(* CoDeSys 2.3 export: SESH_CODESYS.EXP *)
(* Libraries: C:\Program Files (x86)\WAGO Software\CoDeSys V2.3\Targets\WAGO\Libraries\POWER_MEASUREMENT\PowerMeasurement_494_02.lib 7.10.15 13:30:30, Iecsfc.lib 16.5.13 14:00:50, mod_com.lib 16.5.13 14:00:50, Modb_l05.lib 22.4.13 12:50:12, SerComm.lib 16.5.13 14:00:50, Serial_Interface_01.lib 22.4.13 12:50:14, Standard.lib 20.5.14 08:13:26, SYSLIBCALLBACK.LIB 16.5.13 14:00:50, SysLibFile.lib 16.5.13 14:00:50, SysLibSem.lib 16.5.13 14:00:50, SysLibSockets.lib 22.5.14 16:16:32, SysLibTime.lib 16.5.13 14:00:48, Wago_MBCFG_COMMON_01.lib 5.12.13 11:10:18, Wago_MBCFG_SERIAL_01.lib 17.9.14 14:24:36, WagoLibMySQL_03.lib 23.7.14 09:13:36, WagoLibSHA1.lib 19.9.11 08:14:42 *)

(* PLC configuration (modules and I/O channels)
PLC Configuration [Root] node -1, in %IB0 out %QB0
  K-Bus [K_Bus] node 0, in %IB0 out %QB0 {param 201019000 = 1; param 201019001 = 10000; param 201019002 = 0; param 201019003 = 1}
    0750-0652#24 RS-232/RS-485 Interface adjustable (24 Bytes) [Type_30_1_Channels] node 0, in %IB120 out %QB120
      AT %IB0 [BYTEOnB_I] First Byte of 24
      AT %QB0 [BYTEOnB_Q] First Byte of 24
    0750-0652#24 RS-232/RS-485 Interface adjustable (24 Bytes) [Type_30_1_Channels] node 1, in %IB120 out %QB120
      AT %IB24 [BYTEOnB_I] First Byte of 24
      AT %QB24 [BYTEOnB_Q] First Byte of 24
    0750-0652#24 RS-232/RS-485 Interface adjustable (24 Bytes) [Type_30_1_Channels] node 2, in %IB144 out %QB144
      AT %IB48 [BYTEOnB_I] First Byte of 24
      AT %QB48 [BYTEOnB_Q] First Byte of 24
    0750-0494 3-phase PoM480/ 1A [Type_58_1_Channels] node 3, in %IB168 out %QB168
      AT %IW36 [WORDOnW_I] Status Word
      AT %IW37 [WORDOnW_I] Status Word 1
      AT %IW38 [WORDOnW_I] Status Word 2
      AT %IW39 [WORDOnW_I] Status Word 3
      AT %ID20 [DWORDOnD_I] process value 1
      AT %ID21 [DWORDOnD_I] process value 2
      AT %ID22 [DWORDOnD_I] process value 3
      AT %ID23 [DWORDOnD_I] process value 4
      AT %QW36 [WORDOnW_Q] Control Word
      AT %QW37 [WORDOnW_Q] Control Word 1
      AT %QW38 [WORDOnW_Q] Control Word 2
      AT %QW39 [WORDOnW_Q] Control Word 3
    0750-0494 3-phase PoM480/ 1A [Type_58_1_Channels] node 4, in %IB192 out %QB192
      AT %IW48 [WORDOnW_I] Status Word
      AT %IW49 [WORDOnW_I] Status Word 1
      AT %IW50 [WORDOnW_I] Status Word 2
      AT %IW51 [WORDOnW_I] Status Word 3
      AT %ID26 [DWORDOnD_I] process value 1
      AT %ID27 [DWORDOnD_I] process value 2
      AT %ID28 [DWORDOnD_I] process value 3
      AT %ID29 [DWORDOnD_I] process value 4
      AT %QW48 [WORDOnW_Q] Control Word
      AT %QW49 [WORDOnW_Q] Control Word 1
      AT %QW50 [WORDOnW_Q] Control Word 2
      AT %QW51 [WORDOnW_Q] Control Word 3
    0750-0483 2 AI 0-30V DC Differential Measurement Input [Type_8_2_Channels] node 5, in %IB216 out %QB216
      AT %IW60 [WORDOnW_I] Ch_1 Input word
      AT %IW61 [WORDOnW_I] Ch_2 Input word
    0750-0513/0000-0001 2 DO 250V AC 2.0A Rel 2NO (PotFree) [Type_10_2_Channels] node 6, in %IB124 out %QB120
      AT %QX60.0 [BOOLOnX_Q] Ch_1 Digital output
      AT %QX60.1 [BOOLOnX_Q] Ch_2 Digital output
  Modbus variables [PFC200MODBUS] node 1, in %IB0 out %QB0 {param 2010330101 = 1; param 2010330102 = 1; param 2010330201 = 1; param 2010330202 = 502; param 2010330203 = 600; param 2010330301 = 1; param 2010330302 = 502; param 2010330401 = 0; param 2010330402 = 1; param 2010330403 = 5000; param 2010330404 = 0; param 2010330405 = 115200; param 2010330406 = 1; param 2010330407 = 1; param 2010330408 = 0; param 2010330409 = 0}
  Modbus-Master [MB_MASTER] node 2, in %IB0 out %QB0
*)

(* Task configuration *)
TASK MYSQL_Logging (PRIORITY := 29, INTERVAL := T#1s0ms);
Main_logger();
END_TASK
TASK MB_RTU_MASTER_TASK (PRIORITY := 30, INTERVAL := T#5ms);
MBCFG_ModbusSlave();
END_TASK

(* Global variable list: Global_Variables *)
VAR_GLOBAL

	gv_sFilePath: STRING;
	gv_iBuffCounter			:INT := 0; (* counter for  buffer*)
	gv_iBuffPointer			:INT := 0; (* pointer  for  buffer*)
	gv_Buffer					:ARRAY[0..gc_MaxBufferSize] OF DataPoint; (*In memory buffer of failed message attempts*)
	gv_isGenSetON                 :BOOL := FALSE;
	gv_DCGenCycleCount     : INT :=0 ;
	gv_statusRELAY1 AT %QX60.0: BOOL;
	gv_statusRELAY2 AT %QX60.1: BOOL;

END_VAR
VAR_GLOBAL CONSTANT

	(* Site specific variables*)
	gc_iSiteCode: INT := 1000; (*1000 is code for Nyange this needs to be somehow made dynamic and unique for each site*)


	MAX_ROWS : WORD := 30; (* Array size for converted table data *)

	gcMySql_iSqlUpperBound: INT := 29; (* Defines the upper bound of "asSqlStatement",
				used by function blocks "MySql_ExecSql" and "MySql_Query" 
				to provide an SQL statement as "ARRAY [0..UpperBound] OF STRING(Size)".
	*)

	gcMySql_iSqlLength: INT := 370; (* Defines the size in byte of an array element
				of "asSqlStatement", used by function blocks "MySql_ExecSql" and "MySql_Query" 
				to provide an SQL statement as "ARRAY [0..UpperBound] OF STRING(Size)".
	*)
	raw_SQL_STR_LENGTH: INT := 350;

	(* MYSQL configs *)
	gc_sHost : STRING := '### your mysql server address here';  (*'application.dyndns.info';*)
	gc_uiPort : UINT := 3306;
	gc_sUser : STRING := '### your mysql server username ';
	gc_sPwd : STRING := '### your mysql password';
	gc_sDB : STRING := '### your MYSQL database';   	(* Optional - Name of database instance to connect to *)
	gc_sTable:STRING := '### your MYSql table' ;

	(* CSV Writing/Logging parameters*)
	gc_xWriteToSD: BOOL := TRUE;

	iMaxParams			:INT:=5;(* Number of Parameters per File *)
	gc_ParameterCount	:INT:=1;(* Number of Values per Parameter *)
	gc_RawDataSize		:UINT:=500; (* Raw data size for reading in file ASCII *)
	gc_MaxBufferSize 	       :INT := 5000; (*number of items to hold in memory*)
	gc_sFileName		: STRING := 'buffer.csv'; (* Working Filename   Complete path + filename *)

	(* Logging constants*)
	gc_LogInterval             :TIME := T#10s;
	gc_iTotalParams		:INT := 18;

	(* generator constants*)
	gc_DCVoltageGenSetON :REAL := 24; (*make this a bit higher tha load shedding time*)
	gc_DCVoltageGenSetOFF :REAL := 26; (*make this estimate soc %80*)

	(*how many cycles do we wait before we trigger the genset need to calculate based no cycletime *gc_DCGenCycleCount = total_seconds  *)
	gc_DCGenCycleCount       :INT := 40;

END_VAR

(* Data type *)
TYPE DataPoint :
	STRUCT
		(*Common variables*)
		iSiteCode:INT;
		timeStamp: STRING;

		(*AC Variables*)
		rTotalActivePower:REAL;
		rTotalReactivePower:REAL;
		rTotalApparentPower:REAL;
	      rTotalPowerFactorPF:REAL;
		rTotalActiveEnergy:REAL;
		rTotalReactiveEnergy:REAL;
		rTotalApparentEnergy:REAL;
		xRotatingField:BOOL;
		arFrequency_1:REAL;
		arVoltage_L_N_1:REAL;
		arCurrent_1:REAL;
		arFrequency_2:REAL;
		arVoltage_L_N_2:REAL;
		arCurrent_2:REAL;
		arFrequency_3:REAL;
		arVoltage_L_N_3:REAL;
		arCurrent_3:REAL;

		(* DC Variables *)
		DCV1 :REAL;
		DCV2 :REAL;
		DCPower1: REAL;
		DCPower2: REAL;
		DCCurr1 : REAL;
		DCCurr2 : REAL;


		END_STRUCT
END_TYPE

(* Data type *)
TYPE RowData :
  STRUCT
  	dtDt 		: DT; 		(* Table field "timestamp" 	- MySql_Datatype "datetime" 	*)
  	asString 	: ARRAY [0..9] OF STRING(255);	(* Table fields "s0"-"s9" MySql_Datatype "varchar(255)" 	*)
  END_STRUCT
END_TYPE

(* Data type *)
TYPE TableData :
  STRUCT
	xValid : BOOL;
	iRowCount : INT;
	astRow : ARRAY [0..gcMySql_dwMaxRowCount] OF RowData;
  END_STRUCT
END_TYPE

(* Data type *)
TYPE typCSV :
STRUCT
	sDescription	:STRING;
	Parameter		:ARRAY[1..gc_ParameterCount] OF REAL;
END_STRUCT
END_TYPE

(* POU Main_logger, ST *)
PROGRAM Main_logger
VAR
	xDoIt : BOOL;
	wState : WORD; (* Statemachine*)
	oMySql : MySql_Context; (* Used like Structure for keeping login and status information - Do not call it with in your program *)


	(* working data points *)
	arCurrDataPoint : DataPoint;


	hasBufferedItems :  BOOL; (*Flag indicating the status of the buffer *)
	TONInst : TON; (* Sleep timer  *)


	(* Functionblock to contact MySql server *)
	oMySqlLogin : MySql_Login;

	xConnect : BOOL;
	diErrorLogin : DINT;
	sStatusLogin : STRING(500);
	xConnected : BOOL;


	(* Paremeters for 494 power measurement configuration *)
	xEnable							: BOOL:= TRUE;				(* Activates the function block 											II Aktivierung des Bausteins *)
	tCycleTime						: TIME:=t#1s;					(* Cycletime for reading values											II Zykluszeit für das Auslesen der Messwerte *)
	abIn_750_494 AT %IB72 : ARRAY [0..23] OF BYTE;
       abOut_750_494 AT %QB72:  ARRAY [0..23] OF BYTE;
	d750_494                               :  Fb_750_494_AC_Compact_01;  (* local function block instance*)

	(*Genset*)
	gensetINS :GENSETCheck;


	(* Output DC variables *)
	dc_measure : POWER_MEASURMENT_DC;
	DCV1 :REAL;
	DCV2 :REAL;
	DCPower1: REAL;
	DCPower2: REAL;
	DCCurr1 : REAL;
	DCCurr2 : REAL;

	(* Output variables from 494 *)
      bToken							      : BYTE;
	xReady							: BOOL; 						(* Signal that the last read process is finished 							II Anzeige, dass der letzte Lesevorgang abgeschlossen ist*)
	rTotalActivePower					: REAL;						(* Tota lActive Power 														II Wirkleistung gesamt *)
	rTotalReactivePower				: REAL;						(* Total Reactive Power													II Blindleistung gesamt *)
	rTotalApparentPower				: REAL;						(* Total Apparent Power													II Scheinleistung gesamt *)
	rTotalPowerFactorPF				: REAL;						(* Total Power Factor PF 													II Leistungsfaktor_PF gesamt *)
	rTotalActiveEnergy				: REAL;						(* Total Active Energy	 													II Wirkenergie gesamt *)
	rTotalReactiveEnergy				: REAL;						(* Total Reactive Energy 													II Blindenergie gesamt *)
	rTotalApparentEnergy				: REAL;						(* Total Apparent Energy 													II Scheinenergie gesamt *)
	xRotatingField						: BOOL;						(* Rotating Field 															II Drehfeld rechts *)
	arFrequency						: ARRAY[1..3] OF REAL;		(* Frequency																II Frequenz *)
	arVoltage_L_N					: ARRAY[1..3] OF REAL;		(* Voltage L-N 																II Spannung Lx N *)
	arCurrent							: ARRAY[1..3] OF REAL;		(* Current 															   		II Strom *)
	abFeedback						: ARRAY[1..8] OF BYTE;		(*	0   = no Error 															II kein Fehler
																			1   = Invalid values measure ID 										II Einträge MID nicht gültig
																			2   = Timeout
																			3   = Function block not active 										II Baustein nicht aktiv
																			4   = Settings process active (read/write) 							II Parameterbearbeitung aktiv (Lesen/Schreiben)
																			16  = Overflow Value 1
																			32  = Overflow Value 2
																			48  = Overflow Value 1 + Overflow Value 2
																			64  = Overflow Value 3
																			80  = Overflow Value 1 + Overflow Value 3
																			96  = Overflow Value 2 + Overflow Value 3
																			112 = Overflow Value 1 + Overflow Value 2 + Overflow Value 3
																			128 = Overflow Value 4
																			144 = Overflow Value 1 + Overflow Value 4
																			160 = Overflow Value 2 + Overflow Value 4
																			176 = Overflow Value 1 + Overflow Value 2 + Overflow Value 4
																			192 = Overflow Value 3 + Overflow Value 4
																			208 = Overflow Value 1 + Overflow Value 3 + Overflow Value 4
																			224 = Overflow Value 2 + Overflow Value 3 + Overflow Value 4
																			240 = Overflow Value 1 + Overflow Value 2 + Overflow Value 3 + Overflow Value 4*)



	(* Functionblock to process SQL statements who do not return result sets *)
	oMySqlExec1 : MySql_Execute;
	asSqlStatement1 : ARRAY [0..gcMySql_iSqlUpperBound] OF STRING(gcMySql_iSqlLength);
	xExec1 : BOOL;
	diErrorExec1 : DINT;
	sStatusExec1 : STRING(700);

	(*TODO clean this up these might be unnecassar delete if not used *)
	(* Functionblock to process SQL statements who return result sets *)
	oMySqlQuery1 : MySql_Query;
	asSqlQuery1 : ARRAY [0..gcMySql_iSqlUpperBound] OF STRING(gcMySql_iSqlLength);
	xQuery1 : BOOL;
	diErrorQuery1 : DINT;
	sStatusQuery1 : STRING(500);
	stQueryResult1 : MySql_ResultSet;


	(* Convert "stQueryResult" to IEC *)
	stTableData : TableData;
	row, col : INT;
	sValue: STRING(500); (* Returns the value of requested row and col as STRING *)
	dwResult: DWORD; (* Error code of function "MySql_Convert2IEC() *)
	xConvertError : BOOL;

	(* Functionblock to disconnect MySql server *)
	oMySqlLogout : MySql_Logout;
	xDisconnect : BOOL;
	diErrorLogout : DINT;
	sStatusLogout : STRING(500);

	(* Helpers *)
	iHelp : INT;
	i : INT;
	END_: BOOL;
	strTempSQLStatement: STRING(raw_SQL_STR_LENGTH);


	(* debug variables *)
	iCountExecFailed: INT;
	xDolt: BOOL;
END_VAR
(*Get AC power data every cycle*)


d750_494 (						    xEnable:=xEnable,
										tCycleTime:=tCycleTime,
										abOut_750_494:=abOut_750_494,
										abIn_750_494:=abIn_750_494,
										bToken:=bToken,
										xReady=>xReady,
										rTotalActivePower=> rTotalActivePower,
										rTotalReactivePower=>rTotalReactivePower,
										rTotalApparentPower=>rTotalApparentPower,
										rTotalPowerFactorPF=>rTotalPowerFactorPF,
										rTotalActiveEnergy=>rTotalActiveEnergy,
										rTotalReactiveEnergy=>rTotalReactiveEnergy,
										rTotalApparentEnergy=>rTotalApparentEnergy,
										xRotatingField=>xRotatingField,
										arFrequency=>arFrequency,
										arVoltage_L_N=>arVoltage_L_N,
										arCurrent=>arCurrent,
										abFeedback=>abFeedback
										);


(*  Get DC measurement *)
dc_measure(
	tCycleTime:=tCycleTime,
	DCV1=> DCV1,
	DCV2=>DCV2,
	DCPower1=>DCPower1 ,
	DCPower2=>DCPower2,
	DCCurr1=>DCCurr1 ,
	DCCurr2=>DCCurr2 );

(*check genset situation*)
gensetINS(DCBatteryVoltage:=DCV1);

(* Call function block "MySql_Login" every cycle to monitor connection status *)

oMySqlLogin(sHost:= gc_sHost,
			uiPort:= gc_uiPort,
			sUsername:= gc_sUser,
			sPassword:= gc_sPwd,
			sDatabase:=gc_sDB,
			oMySql:= oMySql,
			xStart:= xConnect,
			diError=> diErrorLogin,
			sStatus=> sStatusLogin,
			xConnected=> xConnected);



CASE wState OF
0:

	xConnect := TRUE;
	wState := 10;

10:
	IF xConnected THEN

		xConnect := FALSE;
		IF xRotatingField  THEN  (*  Check that our power measurment model  is ready *)
			wState := 20; (* Proceede to execute SQL*)
		ELSE
			(* this is a different error state *)
			wState:= 45; (* wait and go to holding pattern for power measurement sensor to be ready*)
		END_IF
	ELSE
		wstate:=0;
	END_IF

20: (* prepare sql statement *)
	(*Create data point object to pass around *)
	IF hasBufferedItems THEN
		arCurrDataPoint := gv_Buffer[gv_iBuffPointer];
	ELSE
		arCurrDataPoint := Create_Data_Point (
													iSiteCode:=gc_iSiteCode,
													rTotalActivePower:=rTotalActivePower,
													rTotalReactivePower:=rTotalReactivePower,
													rTotalApparentPower:=rTotalApparentPower,
													rTotalPowerFactorPF:=rTotalPowerFactorPF,
													rTotalActiveEnergy:=rTotalActiveEnergy,
													rTotalReactiveEnergy:=rTotalReactiveEnergy,
													rTotalApparentEnergy:=rTotalApparentEnergy,
													xRotatingField:=xRotatingField,
													arFrequency:=arFrequency,
													arVoltage_L_N:=arVoltage_L_N,
													arCurrent:=arCurrent,
													DCV1 :=DCV1,
													DCV2 :=DCV2,
													DCPower1:= DCPower1,
													DCPower2:= DCPower2,
													DCCurr1 := DCCurr1,
													DCCurr2 :=DCCurr2);
	END_IF
	(* Create AC Statment *)
	asSqlStatement1  := SQLStatement(       toLog     := arCurrDataPoint,
												s_Table:= gc_sTable,
											);


	xExec1 := TRUE; (* Execute SQL-Insert-Statement *)
	wState :=25;

25:
	oMySqlExec1(asSqlCommand:=asSqlStatement1,
					oMySql:=oMySql,
					xStart:=xExec1,
					diError=> diErrorExec1,
					sStatus=>sStatusExec1);

	IF NOT  xExec1 THEN
		(* success *)
			xDisconnect := TRUE;
			wState := 46  (*finished go and disconnect or start again *);
		IF diErrorExec1 = 0 THEN
			IF hasBufferedItems THEN
				IF gv_iBuffCounter = gv_iBuffPointer THEN
					(*Buffer has been cleared reset counters*)
					gv_iBuffCounter := 0;
					gv_iBuffPointer := 0;
					hasBufferedItems := FALSE;
				ELSE
					gv_iBuffPointer := gv_iBuffPointer + 1; (*item pushed was buffered increment pointer *)
				END_IF
			END_IF
		ELSE
			(* Failed *)
			iCountExecFailed := iCountExecFailed +1; (* TODO count number of failures and fire an alarm *)
			wState:=45;
		END_IF
	END_IF


45: (* Wait here to debug convert problem *)
	(* buffer current value into memory *)
	IF gv_iBuffCounter < gc_MaxBufferSize THEN
		gv_Buffer[gv_iBuffCounter] := arCurrDataPoint;
		gv_iBuffCounter := gv_iBuffCounter + 1;
		hasBufferedItems := TRUE; (*Flag indicating the status of the buffer *)
	END_IF
	wState := 46; (*move onto sleep*)

(*sleep X amount of time and continue*)
46:
	TONInst( IN:= TRUE, PT := gc_LogInterval);

	IF TONInst.Q THEN
			wState := 0;
		(* do nothing just wait*)
	END_IF

50: (* Disconnect from database *)
	oMySqlLogout(oMySql:= oMySql,
				 xStart:= xDisconnect,
				 diError=> diErrorLogout,
				 sStatus=> sStatusLogout);
	IF NOT xDisconnect THEN
		xDoIt := FALSE;
		wState := 0;
	END_IF
END_CASE
END_PROGRAM

(* POU External/GENSETCheck, ST *)
FUNCTION_BLOCK GENSETCheck
VAR_INPUT

	DCBatteryVoltage: REAL;
END_VAR
VAR_OUTPUT
END_VAR
VAR
END_VAR
(*Check IF GENSET is already running . IF it is do nothing as battery voltage will increase*)

IF gv_isGenSetON THEN
	(* is batter voltage in a good range *)
	IF DCBatteryVoltage  >  gc_DCVoltageGenSetOFF THEN
		(*IF DC value is below thershold for more then X threshold seconds*)
		IF gc_DCGenCycleCount >= gv_DCGenCycleCount THEN
			(*t rigger dc generator OFF*)
			gv_isGenSetON := FALSE;
			gv_DCGenCycleCount := 0;
		ELSE
			gv_DCGenCycleCount := gv_DCGenCycleCount + 1;
		END_IF

	END_IF

(*check DC (battery) against threshold value*)
ELSIF DCBatteryVoltage < gc_DCVoltageGenSetON THEN
		(*IF DC value is below thershold for more then X threshold seconds*)
		IF gv_DCGenCycleCount >= gc_DCGenCycleCount   THEN
			(*THEN trigger relay to fire GENSET*)
			(*t rigger dc generator OFF*)
			gv_isGenSetON:= TRUE;
			gv_DCGenCycleCount := 0;
		ELSE
			gv_DCGenCycleCount := gv_DCGenCycleCount + 1;
		END_IF

END_IF

gv_statusRELAY1 := gv_isGenSetON;
END_FUNCTION_BLOCK

(* POU POWER_MEASURMENT/POWER_MEASURMENT_DC, ST *)
FUNCTION_BLOCK POWER_MEASURMENT_DC
VAR_INPUT
	tCycleTime						: TIME:=t#1s;					(* Cycletime for reading values*)
END_VAR
VAR_OUTPUT
	DCV1 :REAL;
	DCV2 :REAL;

	DCPower1: REAL;
	DCPower2: REAL;

	DCCurr1 : REAL;
	DCCurr2 : REAL;

END_VAR
VAR
	TONInst : TON; (* Sleep timer  *)
	rDCVoltage1RAW  AT %IW60: WORD;
	rDCVoltage2RAW  AT %IW61 :WORD;

	rDCVoltage1: REAL;
	rDCVoltage2:REAL;

	dcCurrInRaw : INT;
	dcCurrOutRaw :INT;

	dcCurrIn:REAL;
	dcCurrOut:REAL;

	dcReadingError :INT;
END_VAR
TONInst( IN:= TRUE, PT := tCycleTime);

IF TONInst.Q THEN
	(* get sensor reading*)
	MBCFG_ModbusSlave(
		dcCurrIn=>dcCurrInRaw  );

	(* Do conversions from raw numbers to real values smooth with  avereging*)
	dcCurrIn :=  (dcCurrIn + INC_TO_AMPERE(dcCurrInRaw))/2;
	dcCurrOut := INC_TO_AMPERE(dcCurrInRaw);
	
	rDCVoltage1 := (rDCVoltage1 + INC_TO_VOLT(rDCVoltage1RAW))/2;
	rDCVoltage2:= INC_TO_VOLT(rDCVoltage2RAW);

	(* Power Calculations*)
	DCPower1 := (DCPower1 + (dcCurrIn * rDCVoltage1))/2;
	DCPower2 := (dcCurrOut * rDCVoltage2);

	
	DCV1 := rDCVoltage1;
	DCV2 := rDCVoltage2;

	DCCurr1 := dcCurrIn;
	DCCurr2 := dcCurrOut;
	
END_IF
END_FUNCTION_BLOCK

(* POU Generated Code/Serial/MBCFG_ModbusSlave, ST *)
PROGRAM MBCFG_ModbusSlave (* generated by config one prg for each slave *)

VAR_INPUT

END_VAR

VAR_OUTPUT
           dcCurrIn       :    INT;       (**) 


    (*--- system variables (read only) -------------------------*)
    MBCFG_SlaveAddress  :   USINT := 1; (* valid range 1..247   *)
    MBCFG_TimeOut       :   TIME  := t#20ms;
    MBCFG_RequestDelay  :   TIME  := t#0ms; (* 0 means no delay *)
    MBCFG_Error         :   MBCFG_eERROR;
	MBCFG_SERCOM_ERROR  : 	BYTE; (* generated by sercomm.lib -> see documentation of sercomm.lib *)
    (*----------------------------------------------------------*)
END_VAR

{library private}
VAR CONSTANT
    zz_VARIABLECOUNT    :   INT := 1;   (* number of variables  *)
    zz_JOBCOUNT         :   INT := 1;   (* number of jobs       *)
END_VAR
VAR

    (*=== VARIABLE LIST ===============================================================================*)
    zz_VariableList :   ARRAY[1..zz_VARIABLECOUNT] OF MBCFG_typVARIABLE :=
        (   BitSize         := 16,
        ptVar           := 0,
        ReadJobIndex    := 1,
        ReadStartBitNo  := 0,
        WriteJobIndex   := 0,
        WriteStartBitNo := 0 )

                        ;
    (*=================================================================================================*)

    (*=== JOB LIST ====================================================================================*)
    zz_JobList      :   ARRAY[1..zz_JOBCOUNT] OF MBCFG_typCOM_JOB :=
         (   Functioncode            := 3,
        ReadStartAddress        := 4,
        ReadQuantity            := 1,
        WriteStartAddress       := 0,
        WriteQuantity           := 0,
        ptReadData              := 0, 
        ptWriteData             := 0 )

                        ;
    (*=================================================================================================*)

    (*### MODBUS MASTER ##### FIXED CODE ###########################################*)
    zz_MBCFG_MASTER			:	MBCFG_MASTER_SERIAL; (* for serial modbus RTU/ASCII *)
    (*##############################################################################*)

END_VAR
(*--- for each variable one entry ------------------------------------*)
   zz_VariableList[1].ptVar := ADR(dcCurrIn);

(*--------------------------------------------------------------------*)


(*=== call of the master for this slave ====================================================*)
zz_MBCFG_MASTER(   usiSlaveAddress  := MBCFG_SlaveAddress,               (* fixed entry     *)
                    tTimeOut        := MBCFG_TimeOut,                    (* fixed entry     *)
                    iVariableCount  := zz_VARIABLECOUNT,                 (* fixed entry     *)
                    ptVariableList  := ADR(zz_VariableList),             (* fixed entry     *)
                    iJobCount       := zz_JOBCOUNT,                      (* fixed entry     *)
                    ptJobList       := ADR(zz_JobList),                  (* fixed entry     *)
                    tRequestDelay   := MBCFG_RequestDelay,               (* fixed entry     *)
                    MB_ComObject    := MBCFG_COM_OBJECTS.MBCFG_MB_COM_2,(* generated entry *)
                    eError          => MBCFG_Error                       (* fixed entry     *)
                );
(*==========================================================================================*)

MBCFG_SERCOM_ERROR := MBCFG_COM_OBJECTS.MBCFG_MB_COM_2.bInterfaceError;
END_PROGRAM

(* POU Generated Code/Serial/MBCFG/MBCFG_COM_OBJECTS, ST *)
PROGRAM MBCFG_COM_OBJECTS
VAR_INPUT

      MBCFG_MB_COM_2	:	MBCFG_COM_SER_OBJECT := (   ASCII_Mode      := FALSE,
                                                     COM_PORT        := 2,	 
                                                     COM_BAUDRATE    := BAUD_19200,
                                                     COM_PARITY      := PARITY_EVEN,
                                                     COM_STOPBITS    := STOPBITS_1,
                                                     COM_BYTESIZE    := BS_8,
                                                     COM_FLOW_CONTROL:= HALFDUPLEX,
                                                     TIME_OUT        := t#100ms
                                                 );



END_VAR
;
END_PROGRAM

(* POU Helpers/INC_TO_AMPERE, ST *)
FUNCTION INC_TO_AMPERE : REAL
VAR_INPUT
	IN		:	WORD;
END_VAR
(* calculation from increments to ampere *)
INC_TO_AMPERE := (80.0 		(* max. current *)
                                       / 29126)	(* -> 32767 - 3641  Increments of the module for MAX_CURRENT *)
						* WORD_TO_INT(IN);
END_FUNCTION

(* POU Helpers/INC_TO_VOLT, ST *)
FUNCTION INC_TO_VOLT : REAL
VAR_INPUT
	IN		:	WORD;
END_VAR

VAR
	tempVal: REAL;
END_VAR
(* calculation from increments to ampere *)
tempVal := WORD_TO_REAL(IN);

(*divide according to *)
INC_TO_VOLT :=  IN * ( 30.0 / 32767.0);
END_FUNCTION

(* POU Utils/Create_Data_Point, ST *)
FUNCTION Create_Data_Point : DataPoint
VAR
		arCurrDataPoint   : DataPoint;
END_VAR
VAR_INPUT

	iSiteCode: INT;
	rTotalActivePower					: REAL;						(* Tota lActive Power 														II Wirkleistung gesamt *)
	rTotalReactivePower				: REAL;						(* Total Reactive Power													II Blindleistung gesamt *)
	rTotalApparentPower				: REAL;						(* Total Apparent Power													II Scheinleistung gesamt *)
	rTotalPowerFactorPF				: REAL;						(* Total Power Factor PF 													II Leistungsfaktor_PF gesamt *)
	rTotalActiveEnergy				: REAL;						(* Total Active Energy	 													II Wirkenergie gesamt *)
	rTotalReactiveEnergy				: REAL;						(* Total Reactive Energy 													II Blindenergie gesamt *)
	rTotalApparentEnergy				: REAL;						(* Total Apparent Energy 													II Scheinenergie gesamt *)
	xRotatingField						: BOOL;						(* Rotating Field 															II Drehfeld rechts *)
	arFrequency						: ARRAY[1..3] OF REAL;		(* Frequency																II Frequenz *)
	arVoltage_L_N					: ARRAY[1..3] OF REAL;		(* Voltage L-N 																II Spannung Lx N *)
	arCurrent							: ARRAY[1..3] OF REAL;		(* Current 															   		II Strom *)

	(* TODO add the time stamp into buffered items*)

	DCV1 :REAL;
	DCV2 :REAL;

	DCPower1: REAL;
	DCPower2: REAL;

	DCCurr1 : REAL;
	DCCurr2 : REAL;


END_VAR
VAR
END_VAR
	arCurrDataPoint.iSiteCode := iSiteCode;
	arCurrDataPoint.rTotalActivePower :=rTotalActivePower;
	arCurrDataPoint.rTotalReactivePower:=rTotalReactivePower;
	arCurrDataPoint.rTotalApparentPower:=rTotalApparentPower;
	arCurrDataPoint.rTotalPowerFactorPF:=rTotalPowerFactorPF;
	arCurrDataPoint.rTotalActiveEnergy:=rTotalActiveEnergy;
	arCurrDataPoint.rTotalReactiveEnergy:=rTotalReactiveEnergy;
	arCurrDataPoint.xRotatingField:=xRotatingField;


	arCurrDataPoint.arFrequency_1:=arFrequency[1];
	arCurrDataPoint.arVoltage_L_N_1:=arVoltage_L_N[1];
	arCurrDataPoint.arCurrent_1:=arCurrent[1];

	arCurrDataPoint.arFrequency_2:=arFrequency[2];
	arCurrDataPoint.arVoltage_L_N_2:=arVoltage_L_N[2];
	arCurrDataPoint.arCurrent_2:=arCurrent[2];

	arCurrDataPoint.arFrequency_3:=arFrequency[3];
	arCurrDataPoint.arVoltage_L_N_3:=arVoltage_L_N[3];
	arCurrDataPoint.arCurrent_3:=arCurrent[3];

	arCurrDataPoint.timeStamp := Get_Time();

	arCurrDataPoint.DCV1 := DCV1;
	arCurrDataPoint.DCV2:=DCV2;
	arCurrDataPoint.DCPower1:=DCPower1;
	arCurrDataPoint.DCPower2:=DCPower2;
	arCurrDataPoint.DCCurr2:=DCCurr2;
	arCurrDataPoint.DCCurr2:=DCCurr2;


	Create_Data_Point := arCurrDataPoint;
END_FUNCTION

(* POU Utils/Get_Time, ST *)
FUNCTION Get_Time : STRING
VAR_INPUT

END_VAR
VAR
	TimeStamp: STRING;
	SystemTime: SysTime64;
	Time_date: SystemTimeDate;
	TimeDate: CurTimeEx;
	iHours:INT;
	iMinutes:INT;
	iSeconds: INT;
	iDay: INT;
	iMonth: INT;
	iYear: INT;

END_VAR
(* Haal de systeemtijd op *)
TimeDate(SystemTime:= SystemTime, TimeDate:= Time_date);

(* Sla uren en minuten apart op *)
iHours := Time_date.Hour;
iMinutes := Time_date.Minute;
iSeconds := Time_date.Second;
iDay := Time_date.Day;
iMonth := Time_date.Month;
iYear := Time_date.Year;

TimeStamp := CONCAT(TimeStamp,INT_TO_STRING(iYear));
TimeStamp := CONCAT(TimeStamp,INT_TO_STRING(iMonth));
TimeStamp := CONCAT(TimeStamp,INT_TO_STRING(iDay));
TimeStamp := CONCAT(TimeStamp,'T');
TimeStamp := CONCAT(TimeStamp,INT_TO_STRING(iHours));
TimeStamp := CONCAT(TimeStamp,INT_TO_STRING(iMinutes));
TimeStamp := CONCAT(TimeStamp,INT_TO_STRING(iSeconds));
TimeStamp := CONCAT(TimeStamp,'Z');

Get_Time := TimeStamp;
END_FUNCTION

(* POU SQLStatement, ST *)
FUNCTION SQLStatement : ARRAY [0..gcMySql_iSqlUpperBound] OF STRING(gcMySql_iSqlLength)
VAR_INPUT

	toLog:  DataPoint;
	s_Table : STRING;

END_VAR
VAR
	rTotalActivePower					: REAL;						(* Tota lActive Power 														II Wirkleistung gesamt *)
	rTotalReactivePower				: REAL;						(* Total Reactive Power													II Blindleistung gesamt *)
	rTotalApparentPower				: REAL;						(* Total Apparent Power													II Scheinleistung gesamt *)
	rTotalPowerFactorPF				: REAL;						(* Total Power Factor PF 													II Leistungsfaktor_PF gesamt *)
	rTotalActiveEnergy				: REAL;						(* Total Active Energy	 													II Wirkenergie gesamt *)
	rTotalReactiveEnergy				: REAL;						(* Total Reactive Energy 													II Blindenergie gesamt *)
	rTotalApparentEnergy				: REAL;						(* Total Apparent Energy 													II Scheinenergie gesamt *)
	xRotatingField						: BOOL;						(* Rotating Field 															II Drehfeld rechts *)
	arFrequency						: ARRAY[1..3] OF REAL;		(* Frequency																II Frequenz *)
	arVoltage_L_N					: ARRAY[1..3] OF REAL;		(* Voltage L-N 																II Spannung Lx N *)
	arCurrent							: ARRAY[1..3] OF REAL;		(* Current 															   		II Strom *)

	DCV1 :REAL;
	DCV2 :REAL;

	DCPower1: REAL;
	DCPower2: REAL;

	DCCurr1 : REAL;
	DCCurr2 : REAL;

	iSiteCode: INT;

END_VAR
iSiteCode := toLog.iSiteCode;

		(*DC measurement data send *)
		DCV1 := toLog.DCV1 ;
		DCV2 := toLog.DCV2;

		DCPower1:=  toLog.DCPower1;
		DCPower2:=  toLog.DCPower2;
	
		DCCurr1 :=toLog.DCCurr1 ;
		DCCurr2 := toLog.DCCurr2;

		(*AC Daat point *)
		(*TODO time stamp needs to be added if buffered data *)
		rTotalActivePower := toLog.rTotalActivePower;
		rTotalReactivePower := toLog.rTotalReactivePower;
		rTotalApparentPower := toLog.rTotalApparentPower;
		rTotalPowerFactorPF := toLog.rTotalPowerFactorPF;
		rTotalActiveEnergy := toLog.rTotalActiveEnergy;
		rTotalApparentEnergy := toLog.rTotalApparentEnergy;
		xRotatingField := toLog.xRotatingField;
		arFrequency[1] := toLog.arFrequency_1;
		arVoltage_L_N[1] := toLog.arVoltage_L_N_1;
		arCurrent[1] := toLog.arCurrent_1;
		arFrequency[2] := toLog.arFrequency_2;
		arVoltage_L_N[2] := toLog.arVoltage_L_N_2;
		arCurrent[2] := toLog.arCurrent_2;
		arFrequency[3] := toLog.arFrequency_3;
		arVoltage_L_N[3] := toLog.arVoltage_L_N_3;
		arCurrent[3] := toLog.arCurrent_3;
		
		SQLStatement[0] := 'INSERT INTO ';
		SQLStatement[1] := s_Table;
		SQLStatement[2] :=  ' ( rTotalActivePower , rTotalReactivePower , rTotalApparentPower, rTotalPowerFactorPF, rTotalActiveEnergy, rTotalReactiveEnergy, rTotalApparentEnergy,  xRotatingField, arFrequency1 , arFrequency2 ,arFrequency3,arVoltage_L_N1,arVoltage_L_N2, arVoltage_L_N3, arCurrent1,arCurrent2,arCurrent3,DCVolt1,DCVolt2,DCCurr1,DCCurr2 ,DCPower1,DCPower2,iSiteCode)  VALUES ( ';
		(* AC Values *)
		SQLStatement[3] :=  CONCAT(REAL_TO_STRING(rTotalActivePower), ',');
		SQLStatement[4] :=  CONCAT(REAL_TO_STRING(rTotalReactivePower), ',');
		SQLStatement[5] :=  CONCAT(REAL_TO_STRING(rTotalApparentPower), ',');
		SQLStatement[6] :=  CONCAT(REAL_TO_STRING(rTotalPowerFactorPF), ',');
		SQLStatement[7] :=  CONCAT(REAL_TO_STRING(rTotalActiveEnergy), ',');
		SQLStatement[8] :=  CONCAT(REAL_TO_STRING(rTotalReactiveEnergy), ',');
		SQLStatement[9] :=  CONCAT(REAL_TO_STRING(rTotalApparentEnergy), ',');
		SQLStatement[10] :=  CONCAT(BOOL_TO_STRING(xRotatingField), ',');

		SQLStatement[11] :=  CONCAT(REAL_TO_STRING(arFrequency[1]), ',');
		SQLStatement[12] :=  CONCAT(REAL_TO_STRING(arFrequency[2]), ',');
		SQLStatement[13] :=  CONCAT(REAL_TO_STRING(arFrequency[3]), ',');

		SQLStatement[14] :=  CONCAT(REAL_TO_STRING( arVoltage_L_N[1] ), ',');
		SQLStatement[15] :=  CONCAT(REAL_TO_STRING( arVoltage_L_N[2] ), ',');
		SQLStatement[16] :=  CONCAT(REAL_TO_STRING( arVoltage_L_N[3] ), ',');

		SQLStatement[17] :=  CONCAT(REAL_TO_STRING(arCurrent[1] ), ',');
		SQLStatement[18] :=  CONCAT(REAL_TO_STRING(arCurrent[2]), ',');
		SQLStatement[19] :=  CONCAT(REAL_TO_STRING(arCurrent[3]), ',');

		(*  DC Values *)
		SQLStatement[20] :=  CONCAT(REAL_TO_STRING(DCV1), ',');
		SQLStatement[21] :=  CONCAT(REAL_TO_STRING(DCV2), ',');

		SQLStatement[22] :=  CONCAT(REAL_TO_STRING(DCCurr2), ',');
		SQLStatement[23] :=  CONCAT(REAL_TO_STRING(DCCurr2), ',');

		SQLStatement[24] :=  CONCAT(REAL_TO_STRING(DCPower1), ',');
		SQLStatement[25] :=  CONCAT(REAL_TO_STRING(DCPower1), ',');

		SQLStatement[26] :=  CONCAT(INT_TO_STRING(iSiteCode), ' )' );
END_FUNCTION

(* POU Test_Functions/PLC_PRG, ST *)
PROGRAM PLC_PRG
VAR
	rDCVoltage1 : ARRAY [0..23] OF BYTE;
	rDCVoltage2 : ARRAY [0..23] OF BYTE;
END_VAR
DC_TEST();
END_PROGRAM

(* POU Test_Functions/DC_TEST, ST *)
PROGRAM DC_TEST
VAR
	rDCVoltage1  AT %IW60: WORD;
	rDCVoltage2  AT %IW61 :WORD;
	DC1V: REAL;
	DC2V: REAL;
END_VAR
DC1V :=0;
DC2V :=0;
END_PROGRAM

(* POU Configuration/MODBUS_CONFIGURATION, ST *)
PROGRAM MODBUS_CONFIGURATION        
VAR                                
END_VAR                            
(*                                 
   <?xml version="1.0" encoding="UTF-16" standalone="yes"?>
<network xml_structure_version="1">
	<generator_settings minRTUTaskCycleTimeMs="5" minEthaskCycleTimeMs="5" ethSlaveMultiplier="0.1" rtuInterfaceMultiplier="0.1" taskGeneration="true"/>
	<master_interface type="serial" name="Configuration Root Node" com_port="2" baudrate="19200" databits="8" stopbits="1" parity="even" hwtype="RS485" flow_control="Xon/Xoff" asciimode="false" expanded="true">
		<mb_slave comment="" name="ModbusSlave" expanded="true" type="generic">
			<mb_connection type="serial" unitid="1" request_delay_ms="0" response_timeout_ms="20"/>
			<generic_vars comment="" expanded="true">
				<generic_var data_type="INT">
					<generic_params name="dcCurrIn" comment="" expanded="true" mb_access="ro"/>
					<mb_address explicitAccess="false" FCRead="3" FCWrite="0" ReadMBAddress="4" WriteMBAddress="0" ReadBitOffset="0" WriteBitOffset="0"/>
				</generic_var>
			</generic_vars>
		</mb_slave>
	</master_interface>
</network>
                              
*)                                 
;                                  
END_PROGRAM

(* POU POWER_MEASURMENT/POWER_MEASUREMENT_AC, CFC *)
PROGRAM POWER_MEASUREMENT_AC
VAR
	Typ_750_494_State: typ_750_494_State;
	abIn_750_494 AT %IB72 : ARRAY [0..23] OF BYTE;
       abOut_750_494 AT %QB72:  ARRAY [0..23] OF BYTE;
	bToken: BYTE;
	POWER_MEASURE: Fb_750_494_AC_Compact_01;

END_VAR
VAR_OUTPUT
	totalPower: REAL;
	totalReactivePower: REAL;
	totalApparentPower: REAL;
	rotatingField: BOOL;
	totalPowerFactor: REAL;
	totalActiveEnergy: REAL;
	totalReactiveEnergy: REAL;
	totalApparentEnergy: REAL;
	arCurrent: ARRAY [1..3] OF REAL;
	arVoltage: ARRAY [1..3] OF REAL;
	arFrequency: ARRAY [1..3] OF REAL;
	isPowerReady: BOOL;
END_VAR
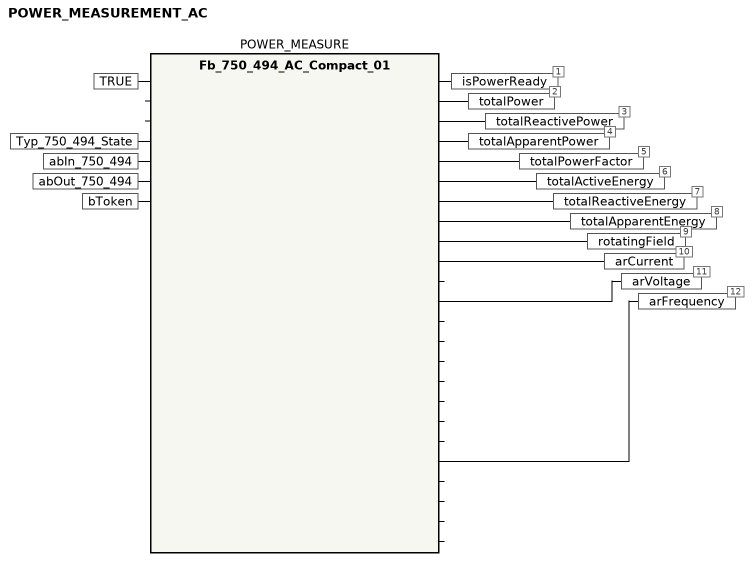
_CFC_ (* Continuous Function Chart, elements in execution order *)
#0 POWER_MEASURE:Fb_750_494_AC_Compact_01(TRUE, -, -, Typ_750_494_State, abIn_750_494, abOut_750_494, bToken)
#1 isPowerReady <= #0.out 1
#2 totalPower <= #0.out 2
#3 totalReactivePower <= #0.out 3
#4 totalApparentPower <= #0.out 4
#5 totalPowerFactor <= #0.out 5
#6 totalActiveEnergy <= #0.out 6
#7 totalReactiveEnergy <= #0.out 7
#8 totalApparentEnergy <= #0.out 8
#9 rotatingField <= #0.out 9
#10 arCurrent <= #0.out 10
#11 arVoltage <= #0.out 12
#12 arFrequency <= #0.out 20
_END_CFC_
END_PROGRAM

(* POU Test_Functions/MYSQL_TEST, ST *)
PROGRAM MYSQL_TEST
VAR

	xDoIt : BOOL;
	wState : WORD; (* Statemachine*)
	oMySql : MySql_Context; (* Used like Structure for keeping login and status information - Do not call it with in your program *)

	sample:BOOL;

	(* Functionblock to contact MySql server *)
	oMySqlLogin : MySql_Login;
	sHost : STRING := 'sesh-dev1.cloudapp.net';  (*'application.dyndns.info';*)
	uiPort : UINT := 3306;
	sUser : STRING := 'wago1';
	sPwd : STRING := 'gle12345';
	sDB : STRING := 'sesh_DB';   	(* Optional - Name of database instance to connect to *)
	sTable:STRING := 'AC_POWER';
	xConnect : BOOL := TRUE;
	diErrorLogin : DINT;
	sStatusLogin : STRING(500);
	xConnected : BOOL;
	iSiteCode: INT := 1000; (*1000 is code for Nyange this needs to be somehow made dynamic and unique for each site*)

END_VAR
(* Call function block "MySql_Login" every cycle to monitor connection status *)
oMySqlLogin(sHost:= sHost,
			uiPort:= uiPort,
			sUsername:= sUser,
			sPassword:= sPwd,
			sDatabase:= sDB,
			oMySql:= oMySql,
			xStart:= xConnect,
			diError=> diErrorLogin,
			sStatus=> sStatusLogin,
			xConnected=> xConnected);


IF xConnected THEN
	sample := TRUE;
	xDoIt := TRUE;
END_IF
END_PROGRAM

(* POU Test_Functions/RELAY_TEST, ST *)
PROGRAM RELAY_TEST
VAR
	wState: BOOL :=FALSE;
	statusRELAY AT %QX60.0: BOOL;
END_VAR
IF NOT wState THEN
		statusRELAY := TRUE;
ELSE
		statusRELAY := FALSE;
END_IF

IF wState THEN
		wState := FALSE;
ELSE
		wState := TRUE;
END_IF
END_PROGRAM

(* POU Utils/ReadCSVFile, ST *)
PROGRAM ReadCSVFile
VAR_INPUT
	sFilename		:STRING;
	bSeperator		:BYTE:=59;(*seperator semicolon:59=;*)
END_VAR
VAR_IN_OUT
	xStart			:BOOL;
	typData			:ARRAY [1..iMaxParams] OF  typCSV;
END_VAR
VAR_OUTPUT
	sStatus			:STRING;
END_VAR
VAR
	bEndOfFile		:BYTE:=13;
	FileIdent		:DWORD;
	rawdata			:ARRAY[0..gc_RawDataSize] OF BYTE;
	filesizev		:DINT;
	tempstring		:STRING;
	startposition	:INT;
	i				:INT;
	j				:INT;
	k				:INT;
END_VAR
IF xStart THEN
	FileIdent:=SysFileOpen(FileName:=sFilename, Mode:='r');
	IF fileident<>0 THEN
		SysFileRead(File:=Fileident, Buffer:=ADR(rawdata), Size:=SIZEOF(rawdata));
		filesizev:=SysFileGetSize(FileName:=sFilename);
		IF filesizev>gc_RawDataSize THEN
			filesizev:=gc_RawDataSize;
		END_IF
		SysFileClose(File:=fileident);(*this function is blocking*)
	ELSE
		sStatus:='File does not exist';
		xStart:=FALSE;
		RETURN;(*no such file available*)
	END_IF
(*copy data to typData array*)
	startposition:=0;
	i:=0;
	FOR j:=1 TO iMaxParams DO
		(*First value in dataset is of type DT. The following value is seperated by bSeperator*)
		WHILE rawdata[startposition+i]<>bSeperator DO
			i:=i+1;
		END_WHILE
		rawdata[startposition+i]:=0;
		MEMCPY(pSourceAddress:=ADR(rawdata[startposition]), pDestinationAddress:=ADR(tempstring), BytesToCopy:=i+1);
		typdata[j].sDescription:=tempstring;
		startposition:=startposition+i+1;
		i:=0;
		(*The parameter values are of type word. The following values are seperated by bSeperator*)
		FOR k:=1 TO gc_ParameterCount-1 DO
			WHILE rawdata[startposition+i]<>bSeperator DO
				i:=i+1;
			END_WHILE
			rawdata[startposition+i]:=0;
			MEMCPY(pSourceAddress:=ADR(rawdata[startposition]), pDestinationAddress:=ADR(tempstring), BytesToCopy:=i+1);
			typdata[j].Parameter[k]:=STRING_TO_REAL(tempstring);
			startposition:=startposition+i+1;
			i:=0;
		END_FOR
		(*Copying the last parameter from typ word. The data set is terminated by CR LF*)
		WHILE rawdata[startposition+i]<>bEndOfFile DO
			i:=i+1;
		END_WHILE
		rawdata[startposition+i]:=0;
		MEMCPY(pSourceAddress:=ADR(rawdata[startposition]), pDestinationAddress:=ADR(tempstring), BytesToCopy:=i+1);
		typdata[j].Parameter[k]:=STRING_TO_REAL(tempstring);
		startposition:=startposition+i+2;(*The data set is terminated by CR LF(13,10)*)
		i:=0;
	END_FOR
(*copy data to typData array finished*)
	sStatus:='Data read OK';
	xStart:=FALSE;
END_IF
END_PROGRAM

(* POU Utils/MEMCPY, ST *)
(*---------------------------------------------------------------------------------------
  WAGO Kontakttechnik GmbH Hansastr. 27 32423 Minden(Westf.) 
  Tel. +49571/887-0 Fax. +49571/887-0                
                                                                                                
  Project: IEC1131 internal library
  
  Function: MEMCPY
  Description: This function copies BytesToCopy bytes from the source
                         address pSourceAddress to the destination address
                         pDestinationAddress
  Date: 25.09.2000

------------------------------------------------------------------------------------------*)
FUNCTION MEMCPY:BOOL
VAR_INPUT
	pSourceAddress:							POINTER TO ARRAY[1..2] OF BYTE;
	pDestinationAddress:						POINTER TO ARRAY[1..2] OF BYTE;
	BytesToCopy:								DINT;
END_VAR
VAR
END_VAR
WHILE (BytesToCopy > 0) DO
	pDestinationAddress^[1]:=pSourceAddress^[1]; (* copy bytes from source to destination *)
	pDestinationAddress:=ADR(pDestinationAddress^[2]); (* increment destination *)
	pSourceAddress:=ADR(pSourceAddress^[2]);(* increment source *)
	BytesToCopy:=BytesToCopy -1; (* decrement number of bytes to copy *)
END_WHILE
END_FUNCTION

(* POU Utils/WriteCSVFile, ST *)
PROGRAM WriteCSVFile
(* 	This function block Writes the contents of the data structure to a CSV File

	Required Libraries:
		Standard.lib
		SysLibFile.lib
*)
VAR_INPUT
	sFILENAME 		:STRING(80); (* Filename to store data to (e.g. 'config.csv' 		*)
	toWrite  			:STRING(500);
	bSeperator		:BYTE :=59;	(* Seperator semicolon:59=;*)
END_VAR
VAR_IN_OUT
	xStart 			:BOOL;	(* Set TRUE to write data, set False to stop.		 *)
END_VAR
VAR_OUTPUT
	sStatus			:STRING;
	iError 			:INT;	(* 00 : Normal Operation	*)
							(* 90 : Can't Open File 	*)
							(* 91 : Can't Close File 	*)
							(* 92 : Can't Write to File 	*)
END_VAR
VAR
	FileOpen		:BOOL := FALSE;
	handle			:DWORD;
	Mode			:STRING[20] := 'rw'; (* read/write *)
	DataString 		:STRING(80);
	i				:INT;
END_VAR
IF xStart THEN
	sStatus := 'Try to open file';
	IF NOT FileOpen THEN
		(* Open File *)
		handle := SysFileOpen(sFileName, Mode);
		IF handle > 0 THEN
			FileOpen := TRUE;
			sStatus := 'File Open OK.';
		ELSE
			iERROR := 90; (* Could not open file. *)
			sStatus := 'Could not open file.';
		END_IF
	END_IF

	IF FileOpen THEN
				IF SysFileWrite(handle, ADR(toWrite), LEN(toWrite)) = 0 THEN
					iERROR := 92; (* Could not write to file *)
					sStatus := 'Could not write file.';
				END_IF
	END_IF

	IF FileOpen THEN
		(* Close file *)
		IF SysFileClose(handle) THEN
			FileOpen := FALSE;
			sStatus := 'File Saved.';
		ELSE
			iERROR := 91; (* Could not close file *)
			sStatus := 'Could not close file.';
		END_IF
		xStart := FALSE;
	END_IF
END_IF
END_PROGRAM

(* POU Utils/Create_Path, ST *)
FUNCTION Create_Path : STRING
VAR_INPUT
END_VAR
VAR
	sFilePath: STRING;
END_VAR
IF gc_xWriteToSD THEN
	sFilePath := '/media/sd/';
ELSE
	sFilePath := '';
END_IF

Create_Path := CONCAT(sFilePath, gc_sFileName);
END_FUNCTION

(* POU Log_to_CSV, ST *)
FUNCTION_BLOCK Log_to_CSV
VAR_INPUT
(*array of data we wish to log to CSV, each data type should be in a seperate CSV?*)
	arToLogData:         ARRAY[1..gc_iTotalParams] OF REAL;

END_VAR
VAR_OUTPUT
END_VAR
VAR
	(*CSV logging variables*)
	(* TODO clean this up removed unused variables*)
	xLoad			: BOOL; (* Initiate load operation *)
	xSave			: BOOL; (* Initiate save operation *)
	sLoadStatus		: STRING; (* Feedback on load *)
	sSaveStatus		: STRING; (* Feedback on save *)
	ConfigData		: ARRAY [1..iMaxParams] OF  typCSV; (* Structure with the config data being loaded or saved *)
	bufferString		:STRING(500);
	bSeperator 		: BYTE := 59; (* Semicolon (;) is the seperator between parameter and value. *)
	iError			: INT; (* Error Code for Save *)

	sFilePath		: STRING; (* SD card is S:\, Internal Path is blank, but this points to the PLC folder *)

	i: INT;
END_VAR
sFilePath := Create_Path();

(* initializse buffer log value *)
bufferString := CONCAT(bufferString , INT_TO_STRING(gv_iBuffCounter) );
bufferString := CONCAT(bufferString , ',' );

(* take the data in array and convert into CSV string format*)
FOR i:=0 TO gc_iTotalParams - 1 DO
	bufferString := CONCAT(bufferString , REAL_TO_STRING(arToLogData[i]));
	bufferString := CONCAT(bufferString , ',' );

	bufferString := CONCAT(bufferString,ASCIIBYTE_TO_STRING(13)); (* CR *)
	bufferString := CONCAT(bufferString,ASCIIBYTE_TO_STRING(10)); (* LF *)

END_FOR
(* function call isn't working right now*)
(*WriteCSVFile(sFilePath,bufferString);*)
gv_iBuffCounter := + 1;
END_FUNCTION_BLOCK

(* POU SPLIT_TO_STR_ARRAY, ST *)
FUNCTION SPLIT_TO_STR_ARRAY : ARRAY [0..gcMySql_iSqlUpperBound] OF STRING(gcMySql_iSqlLength)
VAR_INPUT
	sInputString :      STRING;
	iSizeSplit   :      INT;

END_VAR
VAR

	tempARR: ARRAY [0..gcMysql_iSqlUpperBound] OF STRING(gcMySql_iSqlLength);		(*Temporarry array to merge results	*)
	i: INT := 0;
	iBeginPointer: INT := 0;
	iArraySizeCheck: INT;

END_VAR
(*not using this creatring array maually instead as it doesn't simplify anything*)

iArraySizeCheck := LEN(sInputString) / iSizeSplit; (* We need to see how many slices of the string we will have*)

IF iArraySizeCheck < gcMySql_iSqlUpperBound THEN (* Check that the array we have has enough space to fit these strings*)
	WHILE i  <  gcMysql_iSqlUpperBound  DO
		tempARR[i] := MID( sInputString , iSizeSplit, iBeginPointer);
		i :=  i + 1;
		iBeginPointer := IBeginPointer + iSizeSplit;

	END_WHILE
	SPLIT_TO_STR_ARRAY := tempARR;

END_IF
END_FUNCTION
